// TIA Portal V17 export
// export: Created 2025-06-26T07:49:11.5418644Z, ExportSetting WithDefaults, DisplayName Totally Integrated Automation Portal, DisplayVersion V17 Update 8, DisplayName TIA Portal Openness, DisplayVersion V17 Update 8, DisplayName TIA Portal Version Control Interface, DisplayVersion V17, DisplayName STEP 7 Professional, DisplayVersion V17 Update 8, DisplayName STEP 7 Safety, DisplayVersion V17 Update 6, DisplayName WinCC Advanced, DisplayVersion V17 Update 8
ORGANIZATION_BLOCK "Main"   // OB1, FBD, ProgramCycle
TITLE = "Main Program Sweep (Cycle)"
{ S7_Optimized_Access := 'TRUE' }
VERSION : 0.1
// stored: AutoNumber true, IsIECCheckEnabled false, SetENOAutomatically false
   VAR_INPUT
      Initial_Call : Bool;
      Remanence : Bool;
   END_VAR
BEGIN

REGION Network 1: Land on Mars
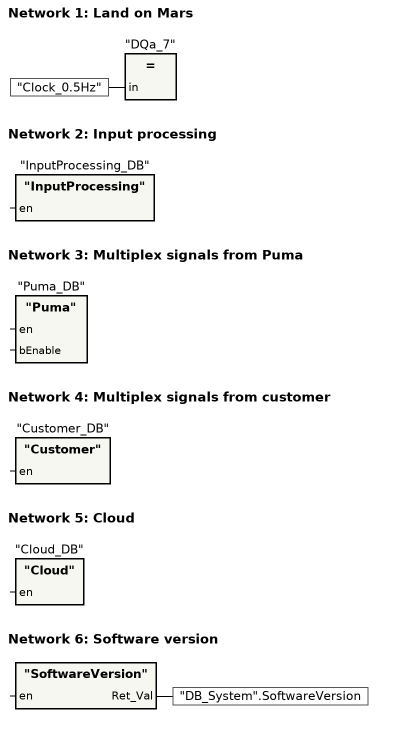
   "DQa_7" := "Clock_0.5Hz";
END_REGION

REGION Network 2: Input processing
   "InputProcessing_DB"();   // "InputProcessing"
END_REGION

REGION Network 3: Multiplex signals from Puma
   "Puma_DB"();   // "Puma"
END_REGION

REGION Network 4: Multiplex signals from customer
   "Customer_DB"();   // "Customer"
END_REGION

REGION Network 5: Cloud
   "Cloud_DB"();   // "Cloud"
END_REGION

REGION Network 6: Software version
   "DB_System".SoftwareVersion := "SoftwareVersion"();
END_REGION
END_ORGANIZATION_BLOCK
